{attribute 'GeneratedUsingTerminal: CU2508--0000'}
{attribute addProperty BoxType "CU2508--0000"}
{attribute addProperty Description "CU2508 Ethernet Port"}
{attribute addProperty Physics "YY"}
{attribute addProperty Id "InfoDataAT %I*InfoData_6F19DB2B2"}
{attribute addProperty CRC "532711307"}
{attribute addProperty Size "2"}
TYPE CU2508_1FC0878B EXTENDS EtcSlaveBoxBase_77A0E4A7 :
STRUCT
	{attribute addProperty Name "InfoData"}
	InfoData : InfoData_6F19DB2B;
END_STRUCT
END_TYPE

(* stored: Version 1.2.0.0, ProductVersion 3.1.4024.11
   DUT CU2508_1FC0878B: Id {666b0cb7-7bf1-4f00-a97c-104aa6ef038c} *)
